FUNCTION_BLOCK FB_Button EXTENDS FB_LinkDevice 
VAR_INPUT
	bEnable		: BOOL; //0-Lamp OFF, 1-Lamp ON
END_VAR

VAR_OUTPUT
	bValue		: BOOL; //0-Released, 1-Pressed
END_VAR

SUPER^();
Control.0 := bEnable;
bValue := Status.0;

END_FUNCTION_BLOCK

(* stored: Version 1.1.0.1, ProductVersion 3.1.4024.12
   POU FB_Button: Id {0326373c-5c67-069e-0e20-ebaf33d35c0e}, SpecialFunc None *)
